Fanuc KAREL source: kf00082.KL

-- PROVISIONAL review KL for V1013-1; original PC SHA256 6b621a07e5d169d21863d8c97ac7fe39dbb8182f80e0ca9e636a9e768bcfb52b
-- Incomplete behavior may be omitted. Consult companion uncertainty JSON. Do not deploy.
PROGRAM KF00082
%NOLOCKGROUP
BEGIN
  -- UNRESOLVED_PC offsets 5-15; opcodes 27,22,31
  -- UNRESOLVED_PC offsets 20-54; opcodes 27,27,2E,22,22,22,22,31
  -- UNRESOLVED_PC offsets 59-93; opcodes 27,22,22,22,22,22,31
  -- UNRESOLVED_PC offsets 98-102; opcodes 7F
END KF00082
